FUNCTION_BLOCK A24_A26 EXTENDS GenericSubarea
VAR_IN_OUT
	spacerRecollector : SpacerRecollectionUnit;
END_VAR
VAR
	robot7 : RobotA26;
	robotSliderA26 : ServoNC;
END_VAR
VAR //sensors to detect spacer on transfer conveyors
	spacerPresent_A24_LRC_C02 AT %I* : BOOL;
	spacerPresent_A24_LRC_C04 AT %I* : BOOL;
	spacerPresent_A24_LRC_C06 AT %I* : BOOL;
	spacerPresent_A24_LRC_C08 AT %I* : BOOL;
	spacerPresent_A24_LRC_C10 AT %I* : BOOL;
	spacerPresent_A24_LRC_C12 AT %I* : BOOL;
END_VAR
VAR
	conveyors : ARRAY[1..6] OF POINTER TO Conveyor;
	step : (IDLE, RECEIVE, MEASURE, SEND, VACANT); //idle, align, active, discharge, complete - replacable with SectionTask enum
	step2 : SectionTask;
END_VAR
(*
A2.4 and A2.6 have interdependent processes
this is a prototype FB that contains the data for both subareas
*)

SUPER^();

CASE step OF
	IDLE:
		allConveyorsRequest(newRequest := ConveyorMode.IDLE);
		
		IF TRUE (*incoming bundle*) THEN
			step := RECEIVE;
		END_IF
		
	RECEIVE:
		allConveyorsRequest(newRequest := ConveyorMode.STOP);
		
		IF TRUE (*area 3 is done transferring*) THEN
			step := MEASURE;
		END_IF
		
	MEASURE:
		
		
	SEND:
		allConveyorsRequest(newRequest := ConveyorMode.FORWARD);
		
		IF allConveyorsVacant() THEN
			step := VACANT;
		END_IF
		
	VACANT:
		allConveyorsRequest(newRequest := ConveyorMode.IDLE);
		step := 0;
		
END_CASE

METHOD PROTECTED allConveyorsRequest : BOOL
VAR_INPUT
	newRequest : ConveyorMode;
END_VAR
VAR
	i : INT;
END_VAR
FOR i:=1 TO 6 BY 1 DO
	conveyors[i]^.setRequest(newRequest := newRequest);
END_FOR
END_METHOD

METHOD PROTECTED allConveyorsVacant : BOOL
VAR_INPUT
END_VAR
VAR
	i : INT;
END_VAR
FOR i:=1 TO 6 BY 1 DO
	IF conveyors[i]^.IsOccupied THEN
		RETURN;
	END_IF
END_FOR

allConveyorsVacant := TRUE;
END_METHOD

METHOD PROTECTED callHardware : BOOL
VAR_INPUT
END_VAR
END_METHOD

METHOD PROTECTED runModules : BOOL
VAR_INPUT
END_VAR
// NETWORK 1
END_METHOD

METHOD PROTECTED setupHardware : BOOL
VAR
	i : INT;
END_VAR
conveyors[1] := ADR(ConveyorSyncUnit.A24_LRC_C02);
conveyors[2] := ADR(ConveyorSyncUnit.A24_LRC_C04);
conveyors[3] := ADR(ConveyorSyncUnit.A24_LRC_C06);
conveyors[4] := ADR(ConveyorSyncUnit.A24_LRC_C08);
conveyors[5] := ADR(ConveyorSyncUnit.A24_LRC_C10);
conveyors[6] := ADR(ConveyorSyncUnit.A24_LRC_C12);
END_METHOD

END_FUNCTION_BLOCK

(* stored: Version 1.1.0.1, ProductVersion 3.1.4024.11
   POU A24_A26: Id {45661656-f465-4c56-89dd-1e9b298b17c5}, SpecialFunc None
   Folder Conveyors: Id {3f427cd1-a7cf-425d-a1ea-6f0b204ca6a0}
   Method allConveyorsRequest: Id {d879df56-0e56-475f-ba6a-6dcdc91dd427}
   Method allConveyorsVacant: Id {324082cd-6db2-4a58-8d6e-68b80ec0f760}
   Method callHardware: Id {e7b7cbec-84f5-4301-8372-5c925f50471f}
   Method runModules: Id {3e067aef-3c96-4d69-9340-7f45388eb0d5}
   Method setupHardware: Id {de28281e-6dde-4862-887a-b60896c5a8c0} *)
